ABB RobotStudio station: FinalSolution.rspag

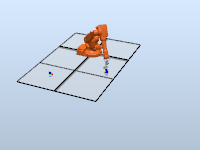
--- station ---
Station FinalSolution (saved by RobotStudio 7.0.8666.559)
Controller IRB_1600_6kg_1.45m
  mechanical unit ROB_1: IRB1600_5_145__01, 6 joints, base frame (0, 0, 0) mm
Layout (positions relative to the parent item):
  - IRB1600_5_145__01 [mechanism, from Robots\IRB1600_5_145__01.rslib] at (0, 0, 0) mm; joint values [-0.8077, 0.9201, 0.0805, 0, 0.5702, -0.8077] (rad or m)
  - Tool4815Final [mechanism, from Libraries\Tool4815Final.rslib] at (712.5, -745, 340.44) mm, rotated rx 180 ry 0 rz 180 deg
Attachment: Tool4815Final is attached to IRB1600_5_145__01 / Link6
Targets, tools, work objects and paths stored in the station and not in the controller backup, written as RAPID:
! task T_ROB1
MODULE Module1
  PROC Path_10()
    MoveL Target_LC_2,v1000,z100,Tool4815Final\WObj:=Workobject_LeftCorner;
  ENDPROC
ENDMODULE


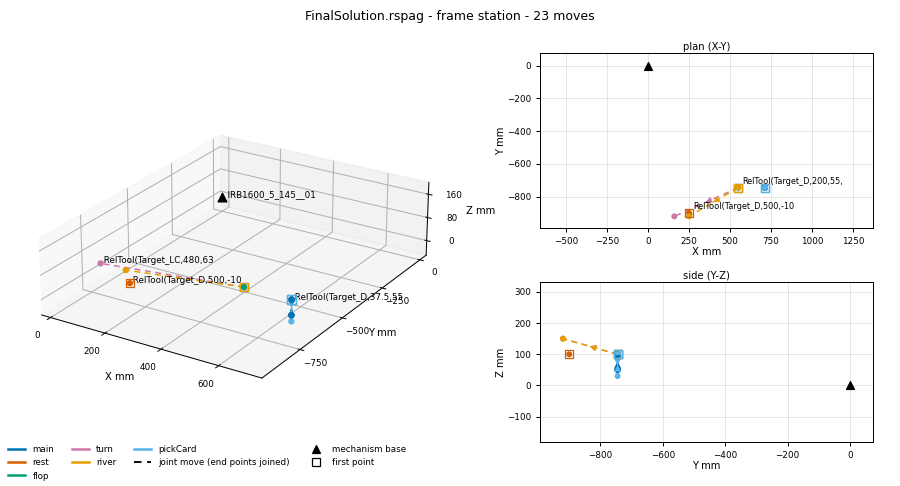
[picture p0: tool path of FinalSolution.rspag in frame station, 23 of 36 moves have a stored position in this frame; points joined in program order, loops and branches not executed]
--- Backups/IRB_1600_6kg_1.45m/RAPID/TASK1/PROGMOD/Module1.mod ---
MODULE Module1
	PERS tooldata Tool4815Final:=[TRUE,[[0,0,240.44],[1,0,0,0]],[0.46438,[0.09,-72.88,36.46],[1,0,0,0],0.003283384,0.001429946,0.00209585]];
	PERS wobjdata Workobject_LeftCorner:=[FALSE,TRUE,"",[[-470,-1400,0],[1,0,0,0]],[[0,0,0],[1,0,0,0]]];
	PERS wobjdata Workobject_Deck:=[FALSE,TRUE,"",[[750,-800,0],[0.707106781,0,0,0.707106781]],[[0,0,0],[1,0,0,0]]];
    !Declaration variables
    VAR socketdev server;
    VAR Socketdev client;
    VAR string message;
    VAR rawbytes data;
    VAR bool Continue;
    VAR bool Continue0;
    VAR bool Continue1;
    VAR bool Continue2;
    VAR bool Continue3;

    !VAR num array{};
    CONST robtarget Target_D:=[[0,0,0],[0,0.707106781,0.707106781,0],[0,0,0,0],[9E+09,9E+09,9E+09,9E+09,9E+09,9E+09]];
    CONST robtarget Target_LC:=[[0,0,0],[0,0.707106781,0.707106781,0],[0,0,0,0],[9E+09,9E+09,9E+09,9E+09,9E+09,9E+09]];
    CONST robtarget Target_LC_2:=[[0,0,0],[0,1,0,0],[0,0,0,0],[9E+09,9E+09,9E+09,9E+09,9E+09,9E+09]];
    !CONST num maxarraysize := 128;
    VAR num array{30};
    !VAR num arraysize:=0;
    !VAR num currentarraysize:=0;
    VAR num Order;

    PROC main()
        SocketCreate server;
        SocketBind server,"192.168.100.100", 55000;
        SocketListen server;
        SocketAccept server, client
                \Time:=WAIT_MAX;
    ! Send a message to the client
        WHILE Continue = FALSE DO
            SocketSend client, \str:="1";
            SocketReceive client,\Rawdata:=data;
            UnpackRawBytes data,1,message,\ASCII:=RawBytesLen(data);
            StringtoNum message,Order;
            IF Order = 0 THEN
                WaitTime 0.1;
            ELSEIF Order = 1 THEN
                 Break;
            ELSEIF Order = 2 THEN
                Continue := TRUE;
            ENDIF
        ENDWHILE

        WHILE Continue0 = FALSE DO
            SocketSend client, \str:="0";
            !Receive a message from the client
            SocketReceive client,\Rawdata:=data;
            UnpackRawBytes data,1,message,\ASCII:=RawBytesLen(data);
            StringtoArray message,array;
            IF message = "" THEN
                WaitTime 0.1;
            ELSE
                Continue0 := TRUE;
            ENDIF
        ENDWHILE


        NoCardFlip;
        MoveJ RelTool(Target_D, 37.5,55, -100),v1000,z100,Tool4815Final\WObj:=Workobject_Deck;
    !Close communication
        !SocketClose server;

   ! FOR k FROM 1 TO 2 DO
        FOR j FROM 1 TO (Dim(array, 1)/2) DO
            IF array{2*j-1} = 2 THEN
                !MoveJ RelTool(Target_D, 37.5,55, -100),v1000,z1,Tool4815Final\WObj:=Workobject_Deck;
                !MoveJ RelTool(Target_D, 37.5,55, -50),v1000,fine,Tool4815Final\WObj:=Workobject_Deck;
                !Suc_suctionCup;
                !MoveJ RelTool(Target_D, 37.5,55, -100),v1000,z1,Tool4815Final\WObj:=Workobject_Deck;
                !MoveJ RelTool(Target_LC,250 ,array{2*i}, -100),v1000,z1,Tool4815Final\WObj:=Workobject_LeftCorner;
                !MoveJ RelTool(Target_LC,250 ,array{2*i}, -50),v1000,fine,Tool4815Final\WObj:=Workobject_LeftCorner;
                !UnSuc_suctionCup;
                !MoveJ RelTool(Target_LC,250 ,array{2*i}, -100),v1000,z1,Tool4815Final\WObj:=Workobject_LeftCorner;

                MoveJ RelTool(Target_D, 37.5,55, -100),v1000,z1,Tool4815Final\WObj:=Workobject_Deck;
                MoveJ RelTool(Target_D, 37.5,55, -50),v1000,fine,Tool4815Final\WObj:=Workobject_Deck;
                Suc_suctionCup;
                MoveJ RelTool(Target_D, 37.5,55, -100),v1000,z1,Tool4815Final\WObj:=Workobject_Deck;
                MoveJ RelTool(Target_LC,250,array{2*j}, -100),v1000,z1,Tool4815Final\WObj:=Workobject_LeftCorner;
                MoveJ RelTool(Target_LC,250,array{2*j}, -50),v1000,fine,Tool4815Final\WObj:=Workobject_LeftCorner;
                UnSuc_suctionCup;
                MoveJ RelTool(Target_LC,250,array{2*j}, -100),v1000,z1,Tool4815Final\WObj:=Workobject_LeftCorner;
            ELSEIF array{2*j-1} = 1 THEN
                !MoveJ RelTool(Target_D, 37.5,55, -100),v1000,z1,Tool4815Final\WObj:=Workobject_Deck;
                !MoveJ RelTool(Target_D, 37.5,55, -50),v1000,fine,Tool4815Final\WObj:=Workobject_Deck;
                !Suc_suctionCup;
                !MoveJ RelTool(Target_D, 37.5, 55, -100),v1000,z1,Tool4815Final\WObj:=Workobject_Deck;
                !MoveJ RelTool(Target_LC, array{2*i},250 ,-100),v1000,z1,Tool4815Final\WObj:=Workobject_LeftCorner;
                !MoveJ RelTool(Target_LC, array{2*i},250 ,-50),v1000,fine,Tool4815Final\WObj:=Workobject_LeftCorner;
                !UnSuc_suctionCup;
                !MoveJ RelTool(Target_LC, array{2*i},250 ,-100),v1000,z1,Tool4815Final\WObj:=Workobject_LeftCorner;

                MoveJ RelTool(Target_D, 37.5,55, -100),v1000,z1,Tool4815Final\WObj:=Workobject_Deck;
                MoveJ RelTool(Target_D, 37.5,55, -50),v1000,fine,Tool4815Final\WObj:=Workobject_Deck;
                Suc_suctionCup;
                MoveJ RelTool(Target_D, 37.5,55, -100),v1000,z1,Tool4815Final\WObj:=Workobject_Deck;
                MoveJ RelTool(Target_LC_2,250, -(array{2*j}),-100),v1000,z1,Tool4815Final\WObj:=Workobject_LeftCorner;
                MoveJ RelTool(Target_LC_2,250, -(array{2*j}),-50),v1000,fine,Tool4815Final\WObj:=Workobject_LeftCorner;
                UnSuc_suctionCup;
                MoveJ RelTool(Target_LC_2,250, -(array{2*j}), -100),v1000,z1,Tool4815Final\WObj:=Workobject_LeftCorner;
           ! ELSEIF array{2*j-1} = 0 THEN
            !   ExitCycle;
            ENDIF
        ENDFOR

        FOR k FROM 1 TO (Dim(array, 1)/2) DO
            IF array{2*k-1} = 2 THEN
                !MoveJ RelTool(Target_D, 37.5,55, -100),v1000,z1,Tool4815Final\WObj:=Workobject_Deck;
                !MoveJ RelTool(Target_D, 37.5,55, -50),v1000,fine,Tool4815Final\WObj:=Workobject_Deck;
                !Suc_suctionCup;
                !MoveJ RelTool(Target_D, 37.5,55, -100),v1000,z1,Tool4815Final\WObj:=Workobject_Deck;
                !MoveJ RelTool(Target_LC,250 ,array{2*i}, -100),v1000,z1,Tool4815Final\WObj:=Workobject_LeftCorner;
                !MoveJ RelTool(Target_LC,250 ,array{2*i}, -50),v1000,fine,Tool4815Final\WObj:=Workobject_LeftCorner;
                !UnSuc_suctionCup;
                !MoveJ RelTool(Target_LC,250 ,array{2*i}, -100),v1000,z1,Tool4815Final\WObj:=Workobject_LeftCorner;

                MoveJ RelTool(Target_D, 37.5,55, -100),v1000,z1,Tool4815Final\WObj:=Workobject_Deck;
                MoveJ RelTool(Target_D, 37.5,55, -50),v1000,fine,Tool4815Final\WObj:=Workobject_Deck;
                Suc_suctionCup;
                MoveJ RelTool(Target_D, 37.5,55, -100),v1000,z1,Tool4815Final\WObj:=Workobject_Deck;
                MoveJ RelTool(Target_LC,250,array{2*k}+100, -100),v1000,z1,Tool4815Final\WObj:=Workobject_LeftCorner;
                MoveJ RelTool(Target_LC,250,array{2*k}+100, -50),v1000,fine,Tool4815Final\WObj:=Workobject_LeftCorner;
                UnSuc_suctionCup;
                MoveJ RelTool(Target_LC,250,array{2*k}+100, -100),v1000,z1,Tool4815Final\WObj:=Workobject_LeftCorner;
            ELSEIF array{2*k-1} = 1 THEN
                !MoveJ RelTool(Target_D, 37.5,55, -100),v1000,z1,Tool4815Final\WObj:=Workobject_Deck;
                !MoveJ RelTool(Target_D, 37.5,55, -50),v1000,fine,Tool4815Final\WObj:=Workobject_Deck;
                !Suc_suctionCup;
                !MoveJ RelTool(Target_D, 37.5, 55, -100),v1000,z1,Tool4815Final\WObj:=Workobject_Deck;
                !MoveJ RelTool(Target_LC, array{2*i},250 ,-100),v1000,z1,Tool4815Final\WObj:=Workobject_LeftCorner;
                !MoveJ RelTool(Target_LC, array{2*i},250 ,-50),v1000,fine,Tool4815Final\WObj:=Workobject_LeftCorner;
                !UnSuc_suctionCup;
                !MoveJ RelTool(Target_LC, array{2*i},250 ,-100),v1000,z1,Tool4815Final\WObj:=Workobject_LeftCorner;

                MoveJ RelTool(Target_D, 37.5,55, -100),v1000,z1,Tool4815Final\WObj:=Workobject_Deck;
                MoveJ RelTool(Target_D, 37.5,55, -50),v1000,fine,Tool4815Final\WObj:=Workobject_Deck;
                Suc_suctionCup;
                MoveJ RelTool(Target_D, 37.5,55, -100),v1000,z1,Tool4815Final\WObj:=Workobject_Deck;
                MoveJ RelTool(Target_LC_2,250, -(array{2*k}+100),-100),v1000,z1,Tool4815Final\WObj:=Workobject_LeftCorner;
                MoveJ RelTool(Target_LC_2,250, -(array{2*k}+100),-50),v1000,fine,Tool4815Final\WObj:=Workobject_LeftCorner;
                UnSuc_suctionCup;
                MoveJ RelTool(Target_LC_2,250, -(array{2*k}+100), -100),v1000,z1,Tool4815Final\WObj:=Workobject_LeftCorner;
            !ELSEIF array{2*k-1} = 0 THEN
            !    ExitCycle;
            ENDIF
       ! ENDFOR
        ENDFOR

        WHILE Continue1 = FALSE DO
            rest;
            SocketSend client, \str:="1";
            SocketReceive client,\Rawdata:=data;
            UnpackRawBytes data,1,message,\ASCII:=RawBytesLen(data);
            StringtoNum message,Order;
            IF Order = 0 THEN
                WaitTime 0.1;
            ELSEIF Order = 1 THEN
                 rest;
                 Break;
            ELSEIF Order = 2 THEN
                flop;
                Continue1 := TRUE;
            ENDIF
        ENDWHILE

        WHILE Continue2 = FALSE DO
            rest;
            SocketSend client, \str:="1";
            SocketReceive client,\Rawdata:=data;
            UnpackRawBytes data,1,message,\ASCII:=RawBytesLen(data);
            StringtoNum message,Order;
            IF Order = 0 THEN
                WaitTime 0.1;
            ELSEIF Order = 1 THEN
                rest;
                Break;
            ELSEIF Order = 2 THEN
                turn;
                Continue2 := TRUE;
            ENDIF
        ENDWHILE

        WHILE Continue3 = FALSE DO
            rest;
            SocketSend client, \str:="1";
            SocketReceive client,\Rawdata:=data;
            UnpackRawBytes data,1,message,\ASCII:=RawBytesLen(data);
            StringtoNum message,Order;
            IF Order = 0 THEN
                WaitTime 0.1;
            ELSEIF Order = 1 THEN
                rest;
                Break;
            ELSEIF Order = 2 THEN
                river;
                Continue3 := TRUE;
            ENDIF
        ENDWHILE
        MoveJ RelTool(Target_D, 37.5,55, -100),v1000,z1,Tool4815Final\WObj:=Workobject_Deck;
    ENDPROC

    PROC StringToArray(string massage, INOUT num Array{*})
        VAR num c1;
        VAR num c2;
        VAR num c3;
        VAR string p1;
        VAR string p2;
        VAR string p3;
        VAR num num1;
        VAR num num2;
        VAR num num3;
        VAR Bool ok;
        VAR Bool strEnd;
        VAR num i;
     !initarray;

        !Store the first number
        c1:= StrFind(message,1,",");
        p1:= StrPart(message,1,c1-1);
        ok:= StrToVal(p1,num1);
        array{1}:=num1;
        !Store the second number
        c2:=StrFind(message, c1+1,",");
        p2:= StrPart(message, c1+1,c2-(c1+1));
        ok:=StrToVal(p2,num2);
        array{2}:=num2;
        !Store the next number
        i := 3;
        WHILE strEnd = FALSE DO
            c3 := StrFind(message,c2+1,",");
            p3:= StrPart(message,c2+1,c3-(c2+1));
            ok:=StrToVal(p3,num3);
            array{i}:=num3;
            i:=i+1;
            c2:=c3;
            IF c2 = StrLen(message) THEN
                strEnd := TRUE;
            ENDIF
        ENDWHILE
    ENDPROC
    PROC Suc_suctionCup()
        !SetDO D652_10_DO1, low;
        WaitTime 1;
    ENDPROC

    PROC UnSuc_suctionCup()
        !SetDO D652_10_DO1, high;
        WaitTime 1;
    ENDPROC

    PROC CardFilp()
        !SetDO D652_10_DO2, High;
        WaitTime 1;
    ENDPROC

    PROC NoCardFlip()
        !SetDO D652_10_DO2, low;
        WaitTime 1;
    ENDPROC

    PROC rest()
        MoveJ RelTool(Target_D, 500,-100, -100),v1000,z1,Tool4815Final\WObj:=Workobject_Deck;
    ENDPROC

    PROC StringtoNum(string massage, INOUT num Order)
        VAR num c1;
        VAR string p1;
        VAR num num1;
        VAR Bool ok;

        c1:= StrFind(message,1,",");
        p1:= StrPart(message,1,c1-1);
        ok:= StrToVal(p1,num1);
        Order := num1;
    ENDPROC


    PROC flop()
        pickCard;
        MoveJ RelTool(Target_D,200 ,55, -100),v1000,fine,Tool4815Final\WObj:=Workobject_Deck;
        UnSuc_suctionCup;
        FOR f FROM 1 TO 3 DO
        pickCard;
        MoveJ RelTool(Target_LC,480,(270+90*f),-150),v1000,fine,Tool4815Final\WObj:=Workobject_LeftCorner;
        CardFilp;
        UnSuc_suctionCup;
        NoCardFlip;
        ENDFOR

    ENDPROC

    PROC turn()
        pickCard;
        MoveJ RelTool(Target_D,200 ,55, -100),v1000,fine,Tool4815Final\WObj:=Workobject_Deck;
        UnSuc_suctionCup;

        pickCard;
        MoveJ RelTool(Target_LC,480,630,-150),v1000,fine,Tool4815Final\WObj:=Workobject_LeftCorner;
        CardFilp;
        UnSuc_suctionCup;
        NoCardFlip;
    ENDPROC

    PROC river()
        pickCard;
        MoveJ RelTool(Target_D,200 ,55, -100),v1000,fine,Tool4815Final\WObj:=Workobject_Deck;
        UnSuc_suctionCup;

        pickCard;
        MoveJ RelTool(Target_LC,480,720,-150),v1000,fine,Tool4815Final\WObj:=Workobject_LeftCorner;
        CardFilp;
        UnSuc_suctionCup;
        NoCardFlip;
    ENDPROC
    !PROC initarray()
    !   currentarraysize:=0;
    !ENDPROC

    !PROC insertelement(num element)
    !  currentarraysize:=currentarraysize+1;
    !  array{currentarraysize}:=element;
    !ENDPROC
    PROC pickCard()
        MoveJ RelTool(Target_D, 37.5,55, -100),v1000,fine,Tool4815Final\WObj:=Workobject_Deck;
        MoveJ RelTool(Target_D, 37.5,55, -30),v1000,fine,Tool4815Final\WObj:=Workobject_Deck;
        Suc_suctionCup;
        WaitTime 0.5;
        MoveJ RelTool(Target_D, 37.5,55, -100),v1000,fine,Tool4815Final\WObj:=Workobject_Deck;
    ENDPROC
ENDMODULE
